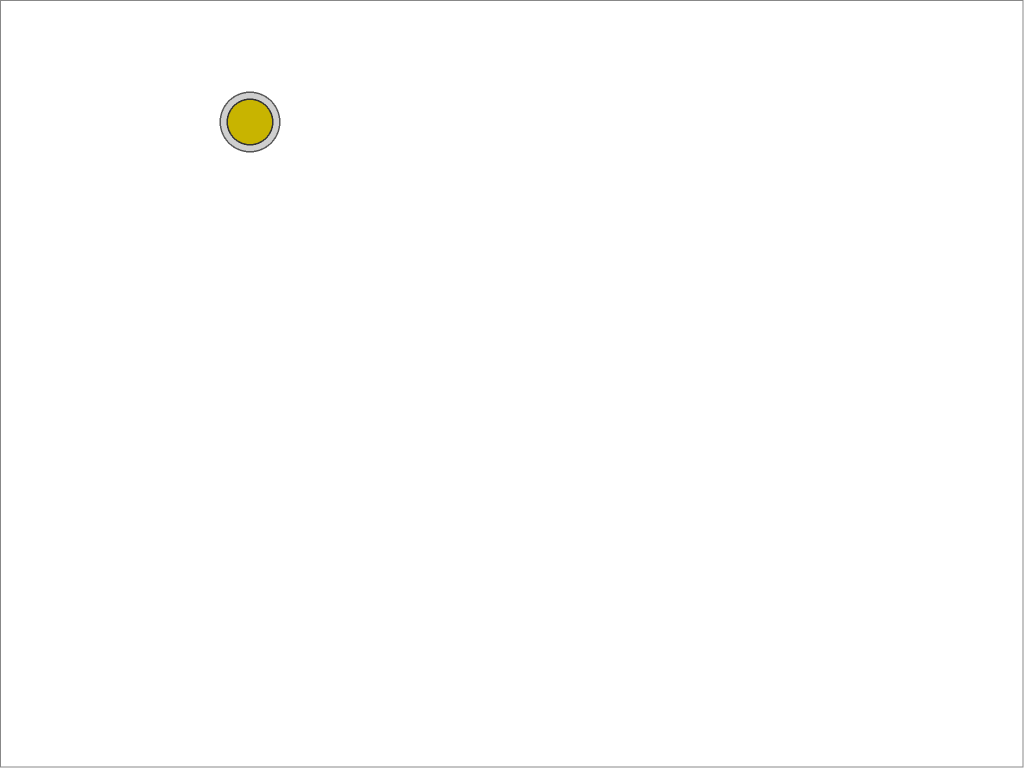
VISUALIZATION HardStuff  // 1024x768
    Lamp1 (215,87 70x70), style: Lamp-Lamp1-Yellow
END_VISUALIZATION

(* stored: Version 1.1.0.1, ProductVersion 3.1.0.19
   Visu HardStuff: Id {135ff5b8-89fb-45d3-a730-de88e6dd09ca} *)
